// TIA Portal V16 export
// export: Created 2020-03-29T18:09:27.7952476Z, ExportSetting None, DisplayName Totally Integrated Automation Portal, DisplayVersion V16 Update 1, DisplayName TIA Portal Version Control Interface, DisplayVersion V16, DisplayName TIA Portal Openness, DisplayVersion V16 Update 1, DisplayName SINAMICS Startdrive Advanced, DisplayVersion V16 Update 1, DisplayName SINAMICS Startdrive G130, G150, S120, S150, SINAMICS MV, S210, DisplayVersion V16 Update 1, DisplayName SINAMICS Startdrive G110M, G120, G120C, G120D, G120P, DisplayVersion V16 Update 1, DisplayName STEP 7 Professional, DisplayVersion V16 Update 1, DisplayName STEP 7 Safety, DisplayVersion V16, DisplayName WinCC Advanced, DisplayVersion V16 Update 1
FUNCTION_BLOCK "Valves"   // FB3, LAD
{ S7_Optimized_Access := 'TRUE' }
// stored: MemoryReserve 100, SetENOAutomatically false
BEGIN
END_FUNCTION_BLOCK
